// TIA Portal V17 export
// export: Created 2023-12-22T15:05:25.308115Z, ExportSetting WithDefaults, DisplayName Totally Integrated Automation Portal, DisplayVersion V17, DisplayName TIA Portal Openness, DisplayVersion V17, DisplayName TIA Portal Version Control Interface, DisplayVersion V17, DisplayName STEP 7 Professional, DisplayVersion V17, DisplayName STEP 7 Safety, DisplayVersion V17, DisplayName WinCC Advanced, DisplayVersion V17
FUNCTION_BLOCK "ELZ"   // FB3, LAD
{ S7_Optimized_Access := 'FALSE' }
VERSION : 0.1
// stored: AutoNumber true, IsIECCheckEnabled false, SetENOAutomatically false, UDAEnableTagReadback false
   VAR_INPUT
      LE : Struct   // Границы датчика
         ST : Bool;   // Общая неисправность
         HH : Bool;   // сработала авария по аварийно высокму уровню
         H : Bool;   // сработало предупреждение по высокому уровню
         L : Bool;   // сработало предупреждение по низкому уровню
         LL : Bool;   // сработало предупрждение по аварийно низкому уровню
         NC : Bool;   // обрыв линии
         SC : Bool;   // короткое замыкание
      END_STRUCT;
      ELZ_Status : Int;   // Статус электролизера
      Pump_Status : Int;   // Статус насоса
      Start_ELZ : Bool;   // Старт электролизера
      Gas_Chanel_1_1 : Bool;   // Датчик загазованности
      Gas_Chanel_1_2 : Bool;   // Датчик загазованности
      Gas_Chanel_2_1 : Bool;   // Датчик загазованности
      Gas_Chanel_2_2 : Bool;   // Датчик загазованности
      KC_1 : Bool;   // Промывочные клапана с фильтров
      KC_2 : Bool;   // Промывочные клапана с фильтров
      AHLS : Bool;   // Верхний аварийный датчик уровня
      Leak : Bool;   // Переполнение поддона
   END_VAR
   VAR_OUTPUT
      ELZ_Start_A : Bool;   // Запуск электролизера
      Pump_Start_A : Bool;   // Запуск насоса
   END_VAR
   VAR DB_SPECIFIC
      Mode : Bool;   // 0 - предупреждение, 1 - остановка через таймер
      Wash : Bool;   // Идет промывка (для панели)
      Gas_Stop : Bool;   // Запрет запуска при загазованности
      Gas : Int;   // Предупреждение о загазованности на панели
      "Step" : Int;
   END_VAR
   VAR
      T_Gas { S7_SetPoint := 'True'} : "Time_M";
      T_ELZ_Start { S7_SetPoint := 'True'} : "Time_M";   // Задержка запуска электролизера
   END_VAR
   // T_ELZ_Start.SP_S := 10;
   VAR_TEMP   // added for the SCL form of the ladder/FBD networks
      _w1 : Bool;
   END_VAR
BEGIN

REGION Network 1: Старт / Выключение электролизера по высокому уровню в баке и по загазованности (порог 2)
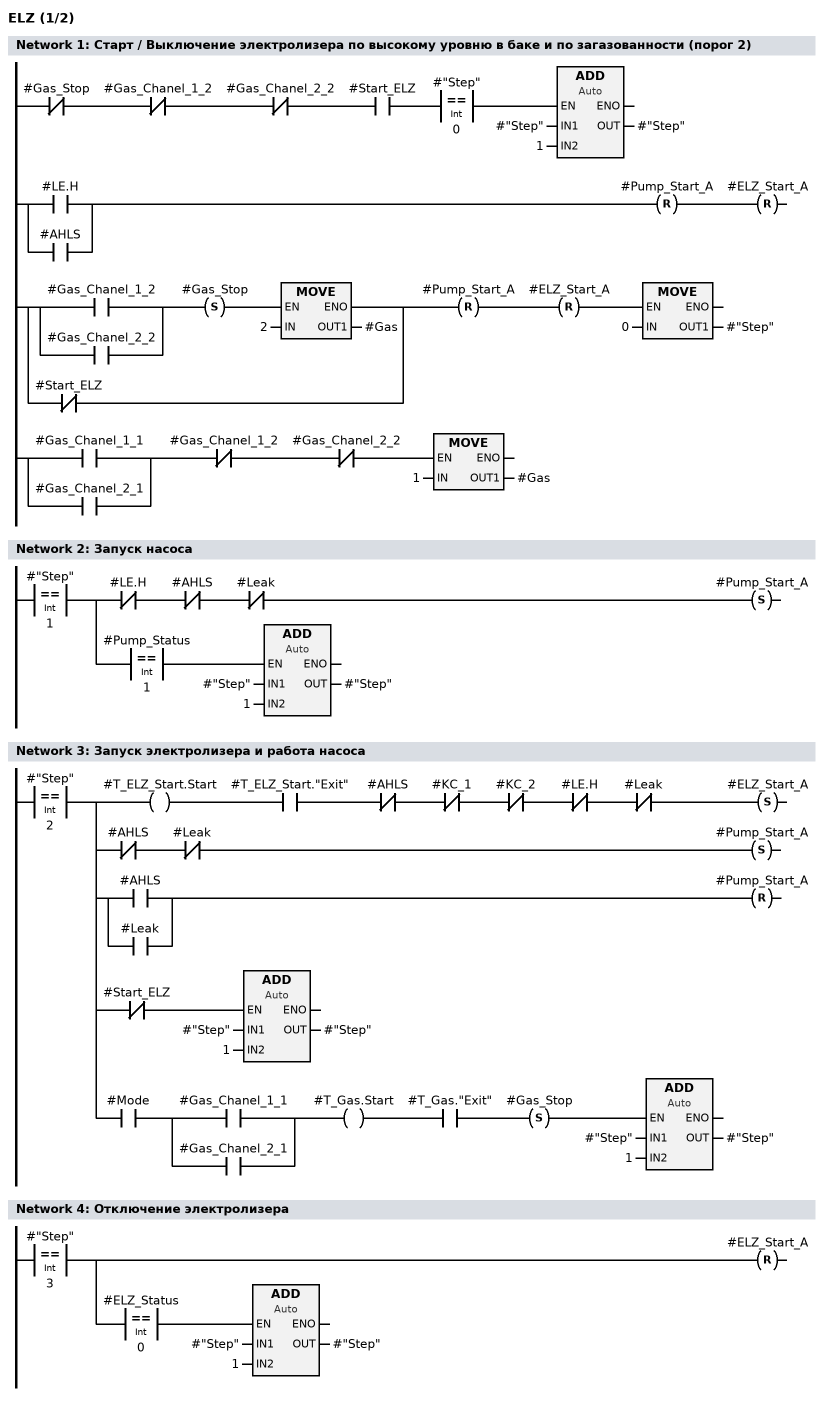
   RUNG wire#powerrail
      I_Contact( #Gas_Stop )
      I_Contact( #Gas_Chanel_1_2 )
      I_Contact( #Gas_Chanel_2_2 )
      Contact( #Start_ELZ )
      { S7_Templates := "SrcType := Int" } EQ_Contact(in1 := #"Step", in2 := 0)
      Add(in1 := #"Step", in2 := 1, out => #"Step")
   END_RUNG
   RUNG wire#powerrail
      Contact( #LE.H )
      wire#w1
      R_Coil( #Pump_Start_A )
      R_Coil( #ELZ_Start_A )
   END_RUNG
   RUNG wire#powerrail
      Contact( #AHLS )
   END_RUNG wire#w1
   RUNG wire#powerrail
      Contact( #Gas_Chanel_1_2 )
      wire#w2
      S_Coil( #Gas_Stop )
      Move(in := 2, out1 => #Gas)
      wire#w3
      R_Coil( #Pump_Start_A )
      R_Coil( #ELZ_Start_A )
      Move(in := 0, out1 => #"Step")
   END_RUNG
   RUNG wire#powerrail
      Contact( #Gas_Chanel_2_2 )
   END_RUNG wire#w2
   RUNG wire#powerrail
      I_Contact( #Start_ELZ )
   END_RUNG wire#w3
   RUNG wire#powerrail
      Contact( #Gas_Chanel_1_1 )
      wire#w4
      I_Contact( #Gas_Chanel_1_2 )
      I_Contact( #Gas_Chanel_2_2 )
      Move(in := 1, out1 => #Gas)
   END_RUNG
   RUNG wire#powerrail
      Contact( #Gas_Chanel_2_1 )
   END_RUNG wire#w4
   // the same network as SCL:
   IF NOT #Gas_Stop AND NOT #Gas_Chanel_1_2 AND NOT #Gas_Chanel_2_2 AND #Start_ELZ AND (#"Step" = 0) THEN
       #"Step" := #"Step" + 1;
   END_IF;
   IF #LE.H OR #AHLS THEN
       #Pump_Start_A := FALSE;
       #ELZ_Start_A := FALSE;
   END_IF;
   #_w1 := #Gas_Chanel_1_2 OR #Gas_Chanel_2_2;
   IF #_w1 THEN
       #Gas_Stop := TRUE;
       #Gas := 2;
   END_IF;
   IF #_w1 OR NOT #Start_ELZ THEN
       #Pump_Start_A := FALSE;
       #ELZ_Start_A := FALSE;
       #"Step" := 0;
   END_IF;
   IF (#Gas_Chanel_1_1 OR #Gas_Chanel_2_1) AND NOT #Gas_Chanel_1_2 AND NOT #Gas_Chanel_2_2 THEN
       #Gas := 1;
   END_IF;
END_REGION

REGION Network 2: Запуск насоса
   RUNG wire#powerrail
      { S7_Templates := "SrcType := Int" } EQ_Contact(in1 := #"Step", in2 := 1)
      wire#w1
      I_Contact( #LE.H )
      I_Contact( #AHLS )
      I_Contact( #Leak )
      S_Coil( #Pump_Start_A )
   END_RUNG
   RUNG wire#w1
      { S7_Templates := "SrcType := Int" } EQ_Contact(in1 := #Pump_Status, in2 := 1)
      Add(in1 := #"Step", in2 := 1, out => #"Step")
   END_RUNG
   // the same network as SCL:
   #_w1 := #"Step" = 1;
   IF #_w1 AND NOT #LE.H AND NOT #AHLS AND NOT #Leak THEN #Pump_Start_A := TRUE; END_IF;
   IF #_w1 AND (#Pump_Status = 1) THEN #"Step" := #"Step" + 1; END_IF;
END_REGION

REGION Network 3: Запуск электролизера и работа насоса
   RUNG wire#powerrail
      { S7_Templates := "SrcType := Int" } EQ_Contact(in1 := #"Step", in2 := 2)
      wire#w1
      Coil( #T_ELZ_Start.Start )
      Contact( #T_ELZ_Start."Exit" )
      I_Contact( #AHLS )
      I_Contact( #KC_1 )
      I_Contact( #KC_2 )
      I_Contact( #LE.H )
      I_Contact( #Leak )
      S_Coil( #ELZ_Start_A )
   END_RUNG
   RUNG wire#w1
      I_Contact( #AHLS )
      I_Contact( #Leak )
      S_Coil( #Pump_Start_A )
   END_RUNG
   RUNG wire#w1
      Contact( #AHLS )
      wire#w2
      R_Coil( #Pump_Start_A )
   END_RUNG
   RUNG wire#w1
      Contact( #Leak )
   END_RUNG wire#w2
   RUNG wire#w1
      I_Contact( #Start_ELZ )
      Add(in1 := #"Step", in2 := 1, out => #"Step")
   END_RUNG
   RUNG wire#w1
      Contact( #Mode )
      wire#w3
      Contact( #Gas_Chanel_1_1 )
      wire#w4
      Coil( #T_Gas.Start )
      Contact( #T_Gas."Exit" )
      S_Coil( #Gas_Stop )
      Add(in1 := #"Step", in2 := 1, out => #"Step")
   END_RUNG
   RUNG wire#w3
      Contact( #Gas_Chanel_2_1 )
   END_RUNG wire#w4
   // the same network as SCL:
   #T_ELZ_Start.Start := #"Step" = 2;
   IF #T_ELZ_Start.Start AND #T_ELZ_Start."Exit" AND NOT #AHLS AND NOT #KC_1 AND NOT #KC_2 AND NOT #LE.H AND NOT #Leak THEN
       #ELZ_Start_A := TRUE;
   END_IF;
   IF #T_ELZ_Start.Start AND NOT #AHLS AND NOT #Leak THEN #Pump_Start_A := TRUE; END_IF;
   IF #T_ELZ_Start.Start AND (#AHLS OR #Leak) THEN #Pump_Start_A := FALSE; END_IF;
   IF #T_ELZ_Start.Start AND NOT #Start_ELZ THEN #"Step" := #"Step" + 1; END_IF;
   #T_Gas.Start := #T_ELZ_Start.Start AND #Mode AND (#Gas_Chanel_1_1 OR #Gas_Chanel_2_1);
   IF #T_Gas.Start AND #T_Gas."Exit" THEN
       #Gas_Stop := TRUE;
       #"Step" := #"Step" + 1;
   END_IF;
END_REGION

REGION Network 4: Отключение электролизера
   RUNG wire#powerrail
      { S7_Templates := "SrcType := Int" } EQ_Contact(in1 := #"Step", in2 := 3)
      wire#w1
      R_Coil( #ELZ_Start_A )
   END_RUNG
   RUNG wire#w1
      { S7_Templates := "SrcType := Int" } EQ_Contact(in1 := #ELZ_Status, in2 := 0)
      Add(in1 := #"Step", in2 := 1, out => #"Step")
   END_RUNG
   // the same network as SCL:
   #_w1 := #"Step" = 3;
   IF #_w1 THEN #ELZ_Start_A := FALSE; END_IF;
   IF #_w1 AND (#ELZ_Status = 0) THEN #"Step" := #"Step" + 1; END_IF;
END_REGION

REGION Network 5: Отключение насоса
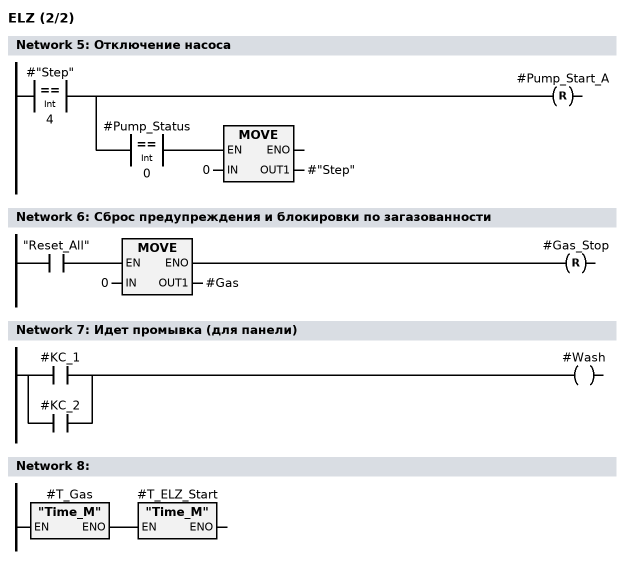
   RUNG wire#powerrail
      { S7_Templates := "SrcType := Int" } EQ_Contact(in1 := #"Step", in2 := 4)
      wire#w1
      R_Coil( #Pump_Start_A )
   END_RUNG
   RUNG wire#w1
      { S7_Templates := "SrcType := Int" } EQ_Contact(in1 := #Pump_Status, in2 := 0)
      Move(in := 0, out1 => #"Step")
   END_RUNG
   // the same network as SCL:
   #_w1 := #"Step" = 4;
   IF #_w1 THEN #Pump_Start_A := FALSE; END_IF;
   IF #_w1 AND (#Pump_Status = 0) THEN #"Step" := 0; END_IF;
END_REGION

REGION Network 6: Сброс предупреждения и блокировки по загазованности
   RUNG wire#powerrail
      Contact( "Reset_All" )
      Move(in := 0, out1 => #Gas)
      R_Coil( #Gas_Stop )
   END_RUNG
   // the same network as SCL:
   IF "Reset_All" THEN
       #Gas := 0;
       #Gas_Stop := FALSE;
   END_IF;
END_REGION

REGION Network 7: Идет промывка (для панели)
   RUNG wire#powerrail
      Contact( #KC_1 )
      wire#w1
      Coil( #Wash )
   END_RUNG
   RUNG wire#powerrail
      Contact( #KC_2 )
   END_RUNG wire#w1
   // the same network as SCL:
   #Wash := #KC_1 OR #KC_2;
END_REGION

REGION Network 8
   RUNG wire#powerrail
      #T_Gas()
      #T_ELZ_Start()
   END_RUNG
   // the same network as SCL:
   #T_Gas(ENO => #_w1);   // "Time_M"
   IF #_w1 THEN
       #T_ELZ_Start();   // "Time_M"
   END_IF;
END_REGION
END_FUNCTION_BLOCK
